INTERFACE I_Call EXTENDS Debug.I_Debug

METHOD Call
VAR_INPUT
	iTag			: Tags.I_Tag;
END_VAR
END_METHOD

END_INTERFACE

(* stored: Version 1.1.0.1
   Itf I_Call: Id {e20aff66-0de3-4f9a-8db1-f7d02b3a4390}
   Method Call: Id {0f557228-c4ae-4503-8235-70a886f9d44f} *)
